FUNCTION F_GetLevelFromPath : UDINT // Get Function nesting level from path by counting '.'
VAR_INPUT
	sPath	: STRING ;
END_VAR
VAR
	sTemp		: STRING ;
	nDotPos		: INT ; 
	nLevel		: UDINT ;
END_VAR

sTemp := sPath ;

REPEAT 
	nDotPos := FIND(sTemp,'.');
	IF nDotPos <> 0 THEN 
		nLevel := nLevel +1 ;
		sTemp := DELETE(STR := sTemp,
						LEN := nDotPos + 1,
						POS	:= 0 );
	END_IF
UNTIL 
	nDotPos = 0	
END_REPEAT

F_GetLevelFromPath := nLevel;

END_FUNCTION

(* stored: Version 1.1.0.1, ProductVersion 3.1.4024.5
   POU F_GetLevelFromPath: Id {4e883c49-73bb-4954-a568-cf4eb5609e00}, SpecialFunc None *)
